Staubli VAL3: getPoint.pgx

public program getPoint(point& x_pPoint[], bool x_bCycle, num x_nIndex)
  local string l_sItem
  local num l_nSize
  local num i
  local num l_nPoint
begin
  // take
  if x_bCycle
    // real point
    x_pPoint=pt:tTraj[sTrajCycle].tData[x_nIndex].pPoint
    if size(x_pPoint)>1
      x_pPoint[1]=pt:tTraj[sTrajCycle].tData[x_nIndex].pCircle
    endIf
  else
    // edit point
    x_pPoint=pEditPoint.tData[x_nIndex].pPoint
    if size(x_pPoint)>1
      x_pPoint[1]=pEditPoint.tData[x_nIndex].pCircle
    endIf
  endIf
end
